// TIA Portal V17 export
// export: Created 2021-12-03T08:13:07.3368427Z, ExportSetting WithDefaults, DisplayName Totally Integrated Automation Portal, DisplayVersion V17, DisplayName TIA Portal Openness, DisplayVersion V17, DisplayName TIA Portal Version Control Interface, DisplayVersion V17, DisplayName STEP 7 Professional, DisplayVersion V17, DisplayName STEP 7 Safety, DisplayVersion V17, DisplayName WinCC Advanced, DisplayVersion V17
DATA_BLOCK "GDB_Simulation"   // DB21
VERSION : 0.1
// stored: AutoNumber false, IsOnlyStoredInLoadMemory false, IsWriteProtectedInAS false
   VAR RETAIN
      DI : Struct
         I_BrLigSrvFlt : Bool;   // Breaker Light and Service Outlet Fault
         I_BrModFlt : Bool;   // Breaker Modulator Fault
         I_BrChilFlt : Bool;   // Breaker Chiller Fault
         I_BrPow1Flt : Bool;   // Breaker Powersupply 1 24VDC Fault
         I_BrPow2Flt : Bool;   // Breaker Powersupply 2 24VDC Fault
         I_BrFrqConvFlt : Bool;   // Breaker Frequnce Converter Conveyor Fault
         I_BrAccConFlt : Bool;   // Breaker Accelerator Console Fault
         I_BrXRayUnitFlt : Bool;   // Breaker X-Ray Unit Fault
         I_BrPowPlcFlt : Bool;   // Breaker Powersupply PS307 (PLC) Fault
         I_SitopPow1Flt : Bool;   // Sitop Diagnose Modul Powersupply 1 Failure
         I_SitopPow2Flt : Bool;   // Sitop Diagnose Modul Powersupply 2 Failure
         I_BrMod1PFlt : Bool;   // Breaker Modulator 230 VAC Fault
         I_Spare1_4 : Bool;   // Spare
         I_Spare1_5 : Bool;   // Spare
         I_Spare1_6 : Bool;   // Spare
         I_Spare1_7 : Bool;   // Spare
         I_Spare2_0 : Bool;   // Spare
         I_Spare2_1 : Bool;   // Spare
         I_Spare2_2 : Bool;   // Spare
         I_Spare2_3 : Bool;   // Spare
         I_Spare2_4 : Bool;   // Spare
         I_Spare2_5 : Bool;   // Spare
         I_Spare2_6 : Bool;   // Spare
         I_Spare2_7 : Bool;   // Spare
         I_P2ConvLocal : Bool;   // Panel 2: Keyswitch Conveyor Local
         "I_/P2ConvLocal" : Bool;   // Panel 2: Keyswitch Conveyor Local (False=Local)
         I_P2ConvFwd : Bool;   // Panel 2: Conveyor move forward
         I_P2ConvBwd : Bool;   // Panel 2: Conveyor move backward
         I_Spare3_4 : Bool;   // Spare
         I_Spare3_5 : Bool;   // Spare
         I_Spare3_6 : Bool;   // Spare
         I_Spare3_7 : Bool;   // Spare
         I_AccStRemMode : Bool;   // Accelerator Status: Remote Mode selected
         I_AccStPowerOn : Bool;   // Accelerator Status: Power on
         I_AccStWarmUp : Bool;   // Accelerator Status: Warming up
         I_AccStClear : Bool;   // Accelerator Status: Clear
         I_AccStReady : Bool;   // Accelerator Status: Ready
         I_AccStXRayOn : Bool;   // Accelerator Status: X-Ray on
         I_AccStFault : Bool;   // Accelerator Status: Fault
         I_AccStNoEmStp : Bool;   // Accelerator Status: Emergency Stop not active
         I_PSConvStpBwd : Bool;   // Photo Sensor Conveyor Stop Position Back
         I_PSConvSlowBwd : Bool;   // Photo Sensor Conveyor Fast Slow Back
         I_PSConvSlowFwd : Bool;   // Photo Sensor Conveyor Fast Slow Front
         I_PSConvStpFwd : Bool;   // Photo Sensor Conveyor Stop Position Front
         I_PSConvXRayBwd : Bool;   // Photo Sensor Conveyor Sensor X-Ray Back
         I_PSConvXRayFwd : Bool;   // Photo Sensor Conveyor Sensor X-Ray Front
         I_Spare5_6 : Bool;   // Spare
         I_Spare5_7 : Bool;   // Spare
         I_ChilVlv_Acc1_Pos : Bool;   // Chiller Valve Position 1
         I_ChilVlv_Acc2_Pos : Bool;   // Chiller Valve Position 2
         I_ModSwch_Acc1_Pos : Bool;   // Modulator Switch Position 1
         I_ModSwch_Acc2_Pos : Bool;   // Modulator Switch Position 2
         I_Spare6_4 : Bool;   // Spare
         I_Spare6_5 : Bool;   // Spare
         I_Spare6_6 : Bool;   // Spare
         I_Spare6_7 : Bool;   // Spare
         I_AccStStandby : Bool;   // Accelerator Status: Standby
         I_AccStMicroWave : Bool;   // Accelerator Status: Microwave (TIS, MIS)
         I_AccStHighDoze : Bool;   // Accelerator Status: High Doze (MIS)
         I_AccStRemouteKey : Bool;   // Accelerator Status: Acc Panel Key
         I_AccStEmStpPanel : Bool;   // Accelerator Status: Emergency Stop Panel (True=No EmStp)
         I_Spare7_5 : Bool;   // Spare
         I_Spare7_6 : Bool;   // Spare
         I_Spare7_7 : Bool;   // Spare
      END_STRUCT;
   END_VAR
BEGIN
END_DATA_BLOCK
